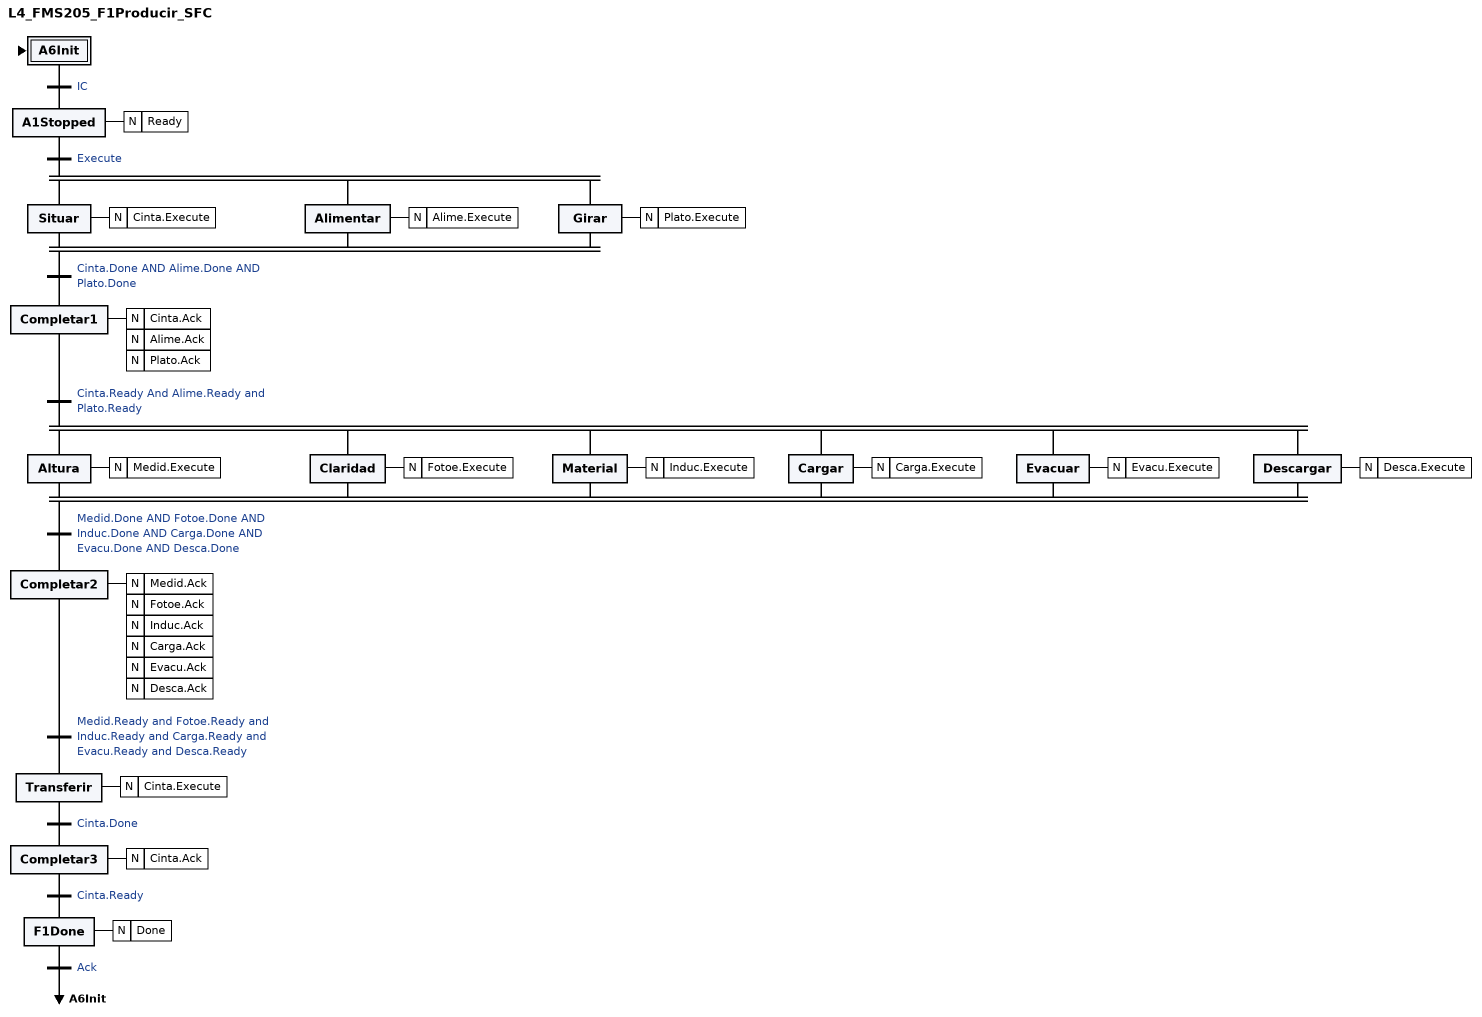
INITIAL_STEP A6Init:
END_STEP
TRANSITION FROM A6Init TO A1Stopped
    := IC;
END_TRANSITION
STEP A1Stopped:
    Ready(N);
END_STEP
TRANSITION FROM A1Stopped TO (Situar, Alimentar, Girar)
    := Execute;
END_TRANSITION
STEP Situar:
    Cinta.Execute(N);
END_STEP
STEP Alimentar:
    Alime.Execute(N);
END_STEP
STEP Girar:
    Plato.Execute(N);
END_STEP
TRANSITION FROM (Situar, Alimentar, Girar) TO Completar1
    := Cinta.Done AND Alime.Done AND Plato.Done;
END_TRANSITION
STEP Completar1:
    Cinta.Ack(N);
    Alime.Ack(N);
    Plato.Ack(N);
END_STEP
TRANSITION FROM Completar1 TO (Altura, Claridad, Material, Cargar, Evacuar, Descargar)
    := Cinta.Ready And Alime.Ready and Plato.Ready;
END_TRANSITION
STEP Altura:
    Medid.Execute(N);
END_STEP
STEP Claridad:
    Fotoe.Execute(N);
END_STEP
STEP Material:
    Induc.Execute(N);
END_STEP
STEP Cargar:
    Carga.Execute(N);
END_STEP
STEP Evacuar:
    Evacu.Execute(N);
END_STEP
STEP Descargar:
    Desca.Execute(N);
END_STEP
TRANSITION FROM (Altura, Claridad, Material, Cargar, Evacuar, Descargar) TO Completar2
    := Medid.Done AND Fotoe.Done AND Induc.Done AND Carga.Done AND Evacu.Done AND Desca.Done;
END_TRANSITION
STEP Completar2:
    Medid.Ack(N);
    Fotoe.Ack(N);
    Induc.Ack(N);
    Carga.Ack(N);
    Evacu.Ack(N);
    Desca.Ack(N);
END_STEP
TRANSITION FROM Completar2 TO Transferir
    := Medid.Ready and Fotoe.Ready and Induc.Ready and Carga.Ready and Evacu.Ready and Desca.Ready;
END_TRANSITION
STEP Transferir:
    Cinta.Execute(N);
END_STEP
TRANSITION FROM Transferir TO Completar3
    := Cinta.Done;
END_TRANSITION
STEP Completar3:
    Cinta.Ack(N);
END_STEP
TRANSITION FROM Completar3 TO F1Done
    := Cinta.Ready;
END_TRANSITION
STEP F1Done:
    Done(N);
END_STEP
TRANSITION FROM F1Done TO A6Init
    := Ack;
END_TRANSITION

END_FUNCTION_BLOCK

// ---- L4 Station Controllers/L4_FMS205_F2SeqPrep_SFC.TcPOU
FUNCTION_BLOCK L4_FMS205_F2SeqPrep_SFC EXTENDS L1_ControllerBase_SFC
// Girar 8 veces el plato para determinar qué tipo de tapa hay en cada sector del plato
VAR_IN_OUT
	Medid			: L3_MedidorTapa;
	Induc		 	: L3_CaptadorInductivo;
	Fotoe			: L3_DetectorFotoelectrico;
	Plato			: L3_PlatoDivisor;
	Tapas			: L6_Tapas;
END_VAR

VAR_OUTPUT
	Seguir 	 		: BOOL;	
	Giros 			: INT;
END_VAR

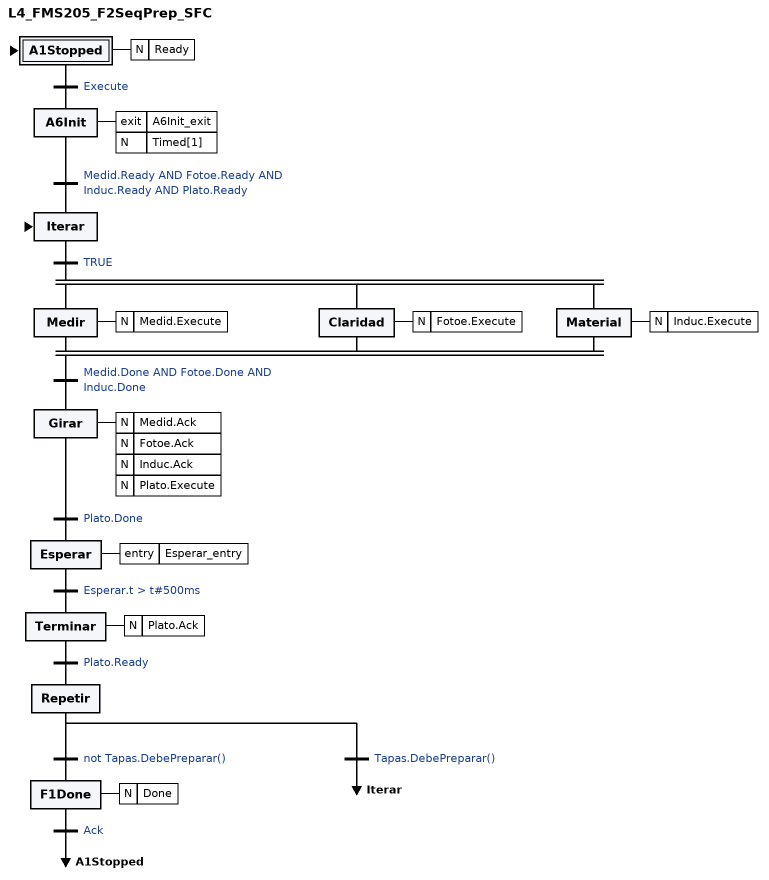
INITIAL_STEP A1Stopped:
    Ready(N);
END_STEP
TRANSITION FROM A1Stopped TO A6Init
    := Execute;
END_TRANSITION
STEP A6Init:
    A6Init_exit(P0);  // exit action
    Timed[1](N);
END_STEP
TRANSITION FROM A6Init TO Iterar
    := Medid.Ready AND Fotoe.Ready AND Induc.Ready AND Plato.Ready;
END_TRANSITION
STEP Iterar:
END_STEP
TRANSITION FROM Iterar TO (Medir, Claridad, Material)
    := TRUE;
END_TRANSITION
STEP Medir:
    Medid.Execute(N);
END_STEP
STEP Claridad:
    Fotoe.Execute(N);
END_STEP
STEP Material:
    Induc.Execute(N);
END_STEP
TRANSITION FROM (Medir, Claridad, Material) TO Girar
    := Medid.Done AND Fotoe.Done AND Induc.Done;
END_TRANSITION
STEP Girar:
    Medid.Ack(N);
    Fotoe.Ack(N);
    Induc.Ack(N);
    Plato.Execute(N);
END_STEP
TRANSITION FROM Girar TO Esperar
    := Plato.Done;
END_TRANSITION
STEP Esperar:
    Esperar_entry(P1);  // entry action
END_STEP
TRANSITION FROM Esperar TO Terminar
    := Esperar.t > t#500ms;
END_TRANSITION
STEP Terminar:
    Plato.Ack(N);
END_STEP
TRANSITION FROM Terminar TO Repetir
    := Plato.Ready;
END_TRANSITION
STEP Repetir:
END_STEP
TRANSITION FROM Repetir TO F1Done
    := not Tapas.DebePreparar();
END_TRANSITION
TRANSITION FROM Repetir TO Iterar
    := Tapas.DebePreparar();
END_TRANSITION
STEP F1Done:
    Done(N);
END_STEP
TRANSITION FROM F1Done TO A1Stopped
    := Ack;
END_TRANSITION

ACTION A6Init_exit:
Giros:=0;
END_ACTION

ACTION Esperar_entry:
Giros:=Giros+1;
END_ACTION

END_FUNCTION_BLOCK

// ---- L4 Station Controllers/L4_FMS205_F3SeqFin_SFC.TcPOU
FUNCTION_BLOCK L4_FMS205_F3SeqFin_SFC EXTENDS L1_ControllerBase_SFC
// Girar 8 veces el plato para determinar qué tipo de tapa hay en cada sector del plato
VAR_INPUT
	TapasOk			: BOOL;
END_VAR

VAR_IN_OUT
	Evacu		 	: L3_Evacuador;
	Plato			: L3_PlatoDivisor;
END_VAR

VAR_OUTPUT
	InitTapas		: BOOL;
	Giros 			: INT := 0;
END_VAR

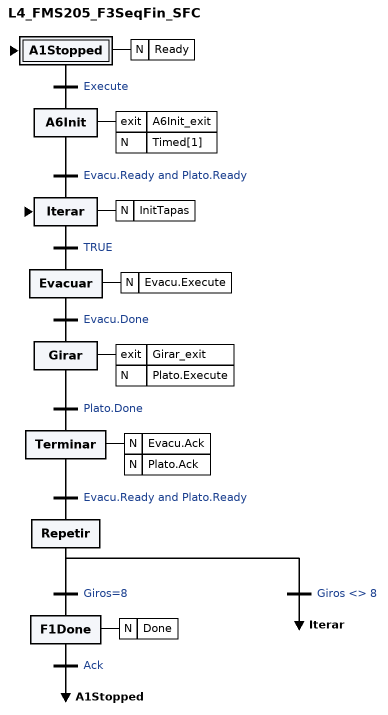
INITIAL_STEP A1Stopped:
    Ready(N);
END_STEP
TRANSITION FROM A1Stopped TO A6Init
    := Execute;
END_TRANSITION
STEP A6Init:
    A6Init_exit(P0);  // exit action
    Timed[1](N);
END_STEP
TRANSITION FROM A6Init TO Iterar
    := Evacu.Ready and Plato.Ready;
END_TRANSITION
STEP Iterar:
    InitTapas(N);
END_STEP
TRANSITION FROM Iterar TO Evacuar
    := TRUE;
END_TRANSITION
STEP Evacuar:
    Evacu.Execute(N);
END_STEP
TRANSITION FROM Evacuar TO Girar
    := Evacu.Done;
END_TRANSITION
STEP Girar:
    Girar_exit(P0);  // exit action
    Plato.Execute(N);
END_STEP
TRANSITION FROM Girar TO Terminar
    := Plato.Done;
END_TRANSITION
STEP Terminar:
    Evacu.Ack(N);
    Plato.Ack(N);
END_STEP
TRANSITION FROM Terminar TO Repetir
    := Evacu.Ready and Plato.Ready;
END_TRANSITION
STEP Repetir:
END_STEP
TRANSITION FROM Repetir TO F1Done
    := Giros=8;
END_TRANSITION
TRANSITION FROM Repetir TO Iterar
    := Giros <> 8;
END_TRANSITION
STEP F1Done:
    Done(N);
END_STEP
TRANSITION FROM F1Done TO A1Stopped
    := Ack;
END_TRANSITION

ACTION A6Init_exit:
Giros:=0;
END_ACTION

ACTION Girar_exit:
Giros:=Giros+1;
END_ACTION

END_FUNCTION_BLOCK

// ---- L4 Station Controllers/L4_FMS205_F6Prueba_SFC.TcPOU
FUNCTION_BLOCK L4_FMS205_F6Prueba_SFC EXTENDS L1_ControllerBase_SFC

VAR_IN_OUT
	Alime			: L3_Alimentador;
	Carga		 	: L3_PickAndPlace;
	Medid			: L3_MedidorTapa;
	Induc		 	: L3_CaptadorInductivo;
	Fotoe			: L3_DetectorFotoelectrico;
	Evacu		 	: L3_Evacuador;
	Desca			: L3_PickAndPlace;
	Plato			: L3_PlatoDivisor;
	Cinta			: L3_Cinta;
END_VAR

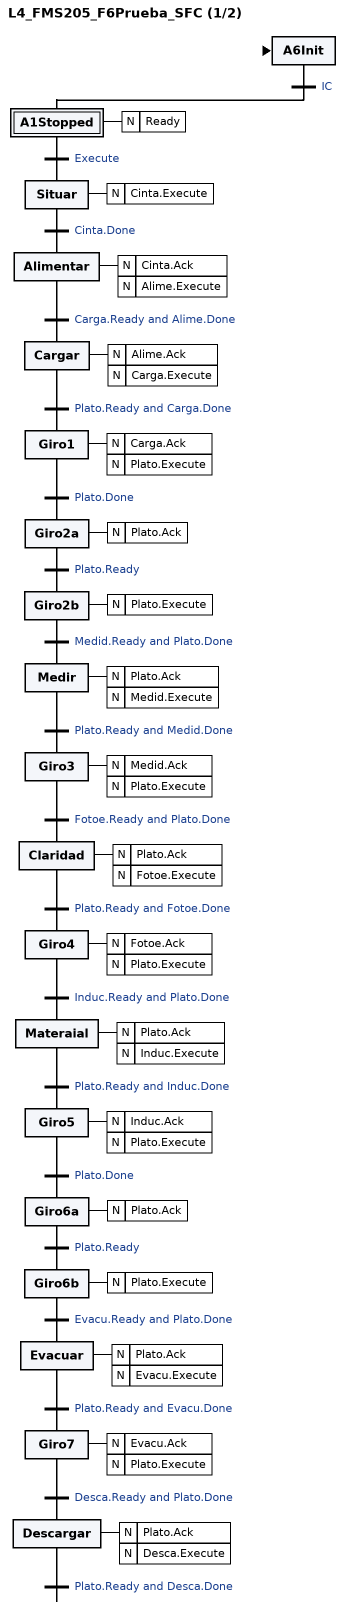
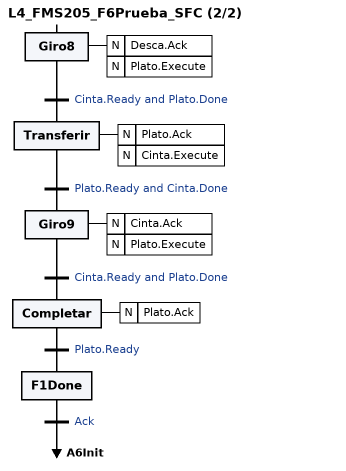
STEP A6Init:
END_STEP
TRANSITION FROM A6Init TO A1Stopped
    := IC;
END_TRANSITION
INITIAL_STEP A1Stopped:
    Ready(N);
END_STEP
TRANSITION FROM A1Stopped TO Situar
    := Execute;
END_TRANSITION
STEP Situar:
    Cinta.Execute(N);
END_STEP
TRANSITION FROM Situar TO Alimentar
    := Cinta.Done;
END_TRANSITION
STEP Alimentar:
    Cinta.Ack(N);
    Alime.Execute(N);
END_STEP
TRANSITION FROM Alimentar TO Cargar
    := Carga.Ready and Alime.Done;
END_TRANSITION
STEP Cargar:
    Alime.Ack(N);
    Carga.Execute(N);
END_STEP
TRANSITION FROM Cargar TO Giro1
    := Plato.Ready and Carga.Done;
END_TRANSITION
STEP Giro1:
    Carga.Ack(N);
    Plato.Execute(N);
END_STEP
TRANSITION FROM Giro1 TO Giro2a
    := Plato.Done;
END_TRANSITION
STEP Giro2a:
    Plato.Ack(N);
END_STEP
TRANSITION FROM Giro2a TO Giro2b
    := Plato.Ready;
END_TRANSITION
STEP Giro2b:
    Plato.Execute(N);
END_STEP
TRANSITION FROM Giro2b TO Medir
    := Medid.Ready and Plato.Done;
END_TRANSITION
STEP Medir:
    Plato.Ack(N);
    Medid.Execute(N);
END_STEP
TRANSITION FROM Medir TO Giro3
    := Plato.Ready and Medid.Done;
END_TRANSITION
STEP Giro3:
    Medid.Ack(N);
    Plato.Execute(N);
END_STEP
TRANSITION FROM Giro3 TO Claridad
    := Fotoe.Ready and Plato.Done;
END_TRANSITION
STEP Claridad:
    Plato.Ack(N);
    Fotoe.Execute(N);
END_STEP
TRANSITION FROM Claridad TO Giro4
    := Plato.Ready and Fotoe.Done;
END_TRANSITION
STEP Giro4:
    Fotoe.Ack(N);
    Plato.Execute(N);
END_STEP
TRANSITION FROM Giro4 TO Materaial
    := Induc.Ready and Plato.Done;
END_TRANSITION
STEP Materaial:
    Plato.Ack(N);
    Induc.Execute(N);
END_STEP
TRANSITION FROM Materaial TO Giro5
    := Plato.Ready and Induc.Done;
END_TRANSITION
STEP Giro5:
    Induc.Ack(N);
    Plato.Execute(N);
END_STEP
TRANSITION FROM Giro5 TO Giro6a
    := Plato.Done;
END_TRANSITION
STEP Giro6a:
    Plato.Ack(N);
END_STEP
TRANSITION FROM Giro6a TO Giro6b
    := Plato.Ready;
END_TRANSITION
STEP Giro6b:
    Plato.Execute(N);
END_STEP
TRANSITION FROM Giro6b TO Evacuar
    := Evacu.Ready and Plato.Done;
END_TRANSITION
STEP Evacuar:
    Plato.Ack(N);
    Evacu.Execute(N);
END_STEP
TRANSITION FROM Evacuar TO Giro7
    := Plato.Ready and Evacu.Done;
END_TRANSITION
STEP Giro7:
    Evacu.Ack(N);
    Plato.Execute(N);
END_STEP
TRANSITION FROM Giro7 TO Descargar
    := Desca.Ready and Plato.Done;
END_TRANSITION
STEP Descargar:
    Plato.Ack(N);
    Desca.Execute(N);
END_STEP
TRANSITION FROM Descargar TO Giro8
    := Plato.Ready and Desca.Done;
END_TRANSITION
STEP Giro8:
    Desca.Ack(N);
    Plato.Execute(N);
END_STEP
TRANSITION FROM Giro8 TO Transferir
    := Cinta.Ready and Plato.Done;
END_TRANSITION
STEP Transferir:
    Plato.Ack(N);
    Cinta.Execute(N);
END_STEP
TRANSITION FROM Transferir TO Giro9
    := Plato.Ready and Cinta.Done;
END_TRANSITION
STEP Giro9:
    Cinta.Ack(N);
    Plato.Execute(N);
END_STEP
TRANSITION FROM Giro9 TO Completar
    := Cinta.Ready and Plato.Done;
END_TRANSITION
STEP Completar:
    Plato.Ack(N);
END_STEP
TRANSITION FROM Completar TO F1Done
    := Plato.Ready;
END_TRANSITION
STEP F1Done:
END_STEP
TRANSITION FROM F1Done TO A6Init
    := Ack;
END_TRANSITION

END_FUNCTION_BLOCK

// ---- L6 Station/L6_FMS205.TcPOU
FUNCTION_BLOCK L6_FMS205 // EXTENDS L1_ModuleBase;

VAR_INPUT
	fbPanel					: L5_Panel := (dr := dr);	
END_VAR

VAR
	// Director, panel y tapas
	dr						: L1_Director;
	tapas					: L6_Tapas;
	
	// módulos de la FMS205
	mdAlimentador			: L3_Alimentador			:= (dr:=dr, ID := 1, Name := 'Alimentador');
	mdPickAndPlaceCarga 	: L3_PickAndPlace			:= (dr:=dr, ID := 2, Name := 'Carga');
	mdMedidorTapa			: L3_MedidorTapa			:= (dr:=dr, ID := 3, Name := 'Medidor');
	mdCaptadorInductivo 	: L3_CaptadorInductivo		:= (dr:=dr, ID := 4, Name := 'Inductivo');
	mdDetectorFotoelectrico : L3_DetectorFotoelectrico	:= (dr:=dr, ID := 5, Name := 'Fotoeléctrico');
	mdEvacuador			 	: L3_Evacuador				:= (dr:=dr, ID := 6, Name := 'Evacuador');
	mdPickAndPlaceDescarga 	: L3_PickAndPlace			:= (dr:=dr, ID := 7, Name := 'Descarga');
	mdPlatoDivisor			: L3_PlatoDivisor			:= (dr:=dr, ID := 8, Name := 'Plato');
	mdCinta					: L3_Cinta					:= (dr:=dr, ID := 9, Name := 'Cinta');
	
	// controladores a nivel estación
	ctrlF1Producir			: L4_FMS205_F1Producir_SFC; 
	ctrlF2SeqPrep			: L4_FMS205_F2SeqPrep_SFC;		
	ctrlF3SeqFin			: L4_FMS205_F3SeqFin_SFC;		
	ctrlF6Prueba			: L4_FMS205_F6Prueba_SFC;
END_VAR

METHOD InitialConditions : BOOL
(* La estación está en condiciones iniciales si cada módulo lo está *)
InitialConditions := (
		mdAlimentador.IC AND
		mdPickAndPlaceCarga.IC AND
		mdMedidorTapa.IC AND 
		mdCaptadorInductivo.IC AND
		mdDetectorFotoelectrico.IC AND
		mdEvacuador.IC AND
		mdPickAndPlaceDescarga.IC AND
		mdPlatoDivisor.IC AND
		mdCinta.IC )  OR dr.gmLocalHost;
END_METHOD

METHOD IsFailied : BOOL
VAR
	NumError	: UDINT;
	Mensaje		: string;
END_VAR
IsFailied:=TRUE;	
IF dr.gmModeActual = L1_GEMMA.A6Inicializando THEN
	IsFailied:=FALSE;
	ManageErrors();
ELSIF dr.gmModeActual = L1_GEMMA.A5PreparandoTrasFallo OR dr.gmModeActual=L1_GEMMA.D2TratamientoFallos THEN
	IF mdAlimentador.fbController.NumError <> 0 THEN
		Mensaje := 'Fallo en alimentador, error=';
		NumError :=	mdAlimentador.fbController.NumError;
		
	ELSIF mdPickAndPlaceCarga.fbController.NumError <> 0 THEN
		Mensaje := 'Fallo en brazo de carga, error=';
		NumError := mdPickAndPlaceCarga.fbController.NumError; 
		
	ELSIF mdMedidorTapa.fbController.NumError <> 0 THEN
		Mensaje := 'Fallo en medidor de altura, error=';
		NumError := mdMedidorTapa.fbController.NumError;
		
	ELSIF mdDetectorFotoelectrico.fbController.NumError <> 0 THEN
		Mensaje := 'Fallo en detector fotoeléctrico, error=';
		NumError := mdDetectorFotoelectrico.fbController.NumError;
		
	ELSIF mdCaptadorInductivo.fbController.NumError<>0 THEN
		Mensaje := 'Fallo en captador inductivo, error=';
		NumError := mdCaptadorInductivo.fbController.NumError;
	
	ELSIF mdEvacuador.fbController.NumError <> 0 THEN
		Mensaje := 'Fallo en evacuador, error=';
		NumError := mdEvacuador.fbController.NumError;
		
	ELSIF  mdPickAndPlaceDescarga.fbController.NumError <> 0 THEN
		Mensaje := 'Fallo en brazo de descarga, error=';
		NumError := mdPickAndPlaceDescarga.fbController.NumError;
		
	ELSIF mdPlatoDivisor.fbController.NumError <> 0 THEN
		Mensaje := 'Fallo en plato giratorio, error=';
		NumError := mdPlatoDivisor.fbController.NumError;
		
	ELSIF mdCinta.fbController.NumError <> 0 THEN
		Mensaje := 'Fallo en cinta, error=';
		NumError := mdCinta.fbController.NumError;
	
	ELSE
		fbPanel.swMensaje := '';
		IsFailied := FALSE;
	END_IF
	
	IF IsFailied THEN
		fbPanel.swMensaje := CONCAT(Mensaje, TO_STRING(NumError));
	END_IF

ELSE
	IsFailied:=FALSE;		
END_IF
END_METHOD

METHOD IsPaused : BOOL
VAR_INPUT
END_VAR
IsPaused := 
		mdAlimentador.fbController.IsPaused() AND
		mdPickAndPlaceCarga.fbController.IsPaused() AND
		mdMedidorTapa.fbController.IsPaused() AND 
		mdCaptadorInductivo.fbController.IsPaused() AND
		mdDetectorFotoelectrico.fbController.IsPaused() AND
		mdEvacuador.fbController.isPaused() AND
		mdPickAndPlaceDescarga.fbController.IsPaused() AND
		mdPlatoDivisor.fbController.IsPaused() AND
		mdCinta.fbController.IsPaused(); (* AND
		ctrlF1Producir.IsPaused() AND
		ctrlF2SeqPrep.IsPaused() AND
		ctrlF3SeqFin.IsPaused() AND
		ctrlF6Prueba.IsPaused();*)
END_METHOD

METHOD ManageErrors : BOOL
mdAlimentador.fbController.ResetError();
mdAlimentador.fbController.ResetError();
mdPickAndPlaceCarga.fbController.ResetError();
mdMedidorTapa.fbController.ResetError();
mdCaptadorInductivo.fbController.ResetError();
mdDetectorFotoelectrico.fbController.ResetError();
mdEvacuador.fbController.ResetError();
mdPickAndPlaceDescarga.fbController.ResetError();
mdPlatoDivisor.fbController.ResetError();
mdCinta.fbController.ResetError();
ctrlF1Producir.ResetError();
ctrlF2SeqPrep.ResetError();
ctrlF3SeqFin.ResetError();
ctrlF6Prueba.ResetError();
END_METHOD

METHOD ProcessCycle : BOOL
// calcular consignas en función del panel y del modo Gemma
dr.Failure 									:= IsFailied();
fbPanel.ProcessCycle(dr:=dr, gmModeActual := dr.gmModeActual, tmReinicio := dr.tmTiempoReinicio);
dr.ProcessCycle(); 

// ejecutar el ciclo de cada Grafcet a nivel estación
ctrlF1Producir.ProcessCycle(dr.gmModeActual);					
ctrlF2SeqPrep.ProcessCycle(dr.gmModeActual);
ctrlF3SeqFin.ProcessCycle(dr.gmModeActual);
ctrlF6Prueba.ProcessCycle(dr.gmModeActual);

// decidir qué tiene que hacer cada módulo
mdAlimentador.Alimentar					:= NOT dr.EndBatch AND NOT tapas.EstaAlimentada; // mdAlimentador.TapaAlimentada;
mdPickAndPlaceCarga.Mover				:= NOT dr.EndBatch AND tapas.EstaAlimentada AND tapas.PuedeCargar(); //  mdAlimentador.TapaAlimentada 
//IF mdPickAndPlaceCarga.TapaMovida THEN
	//mdAlimentador.TapaAlimentada		:= FALSE;
	//tapas.EstaAlimentada				:= FALSE;
	//mdPickAndPlaceCarga.TapaMovida		:= FALSE;	
//END_IF

mdMedidorTapa.Medir						:= tapas.DebeMedir();
mdEvacuador.Evacuar						:= tapas.PuedeEvacuar(gmMode:=dr.gmModeActual);
mdPickAndPlaceDescarga.Mover			:= NOT dr.EndBatch AND mdCinta.Carro_Situado AND tapas.PuedeDescargar();
//IF mdPickAndPlaceDescarga.TapaMovida THEN
	//mdCinta.TapaDescargada				:= TRUE;
	//mdCinta.Transferir					:= TRUE;
	//mdPickAndPlaceDescarga.TapaMovida	:= FALSE;
//END_IF


// controlar el flujo a nivel de la estación
CASE dr.gmModeActual OF
	L1_GEMMA.A1ParadaInicial:						// esperar a que se pida hacer altgo
		dr.EndCycle	:= FALSE;
		dr.EndBatch	:= FALSE;		

	//L1_GEMMA.A3ParadaEstado: 						// esperar la puesta en marcha o reanudar tras parada		
	//L1_GEMMA.A4ParadaObtenida:
	//	dr.IsPaused := IsPaused(); 

	L1_GEMMA.A5PreparandoTrasFallo:
		ManageErrors();		

	L1_GEMMA.A6Inicializando:
		dr.Failure						:= FALSE;
		dr.IsPaused						:= FALSE;
		dr.IC							:= InitialConditions();
		tapas.Inicializar();		
		
	L1_GEMMA.D1ParadaEmergencia:
		dr.IC							:= FALSE;	// obliga a ejecutar la inicialización
		
	L1_GEMMA.D2TratamientoFallos:					// esperar a que el usuario arregle el error
		dr.Failure 		:= IsFailied(); 			// redundante. ManageErrors(); ?
		
	L1_GEMMA.F1ProduccionNormal,
	L1_GEMMA.A2ParaFinCiclo:
		ctrlF1Producir.IC 				:= InitialConditions();
		dr.EndCycle 					:= ctrlF1Producir.Done;
		IF ctrlF1Producir.Done THEN
			dr.EndCycle					:= TRUE;
			dr.cnA3_Estado				:= dr.cnA2_FinCiclo;
			ctrlF1Producir.Execute		:= FALSE;
			ctrlF1Producir.Ack			:= TRUE;			
			dr.EndBatch 				:= tapas.ResReal >= tapas.ReqNumero;			
		ELSIF ctrlF1Producir.Ready AND NOT dr.EndCycle THEN
			dr.EndCycle					:= FALSE;
			ctrlF1Producir.Execute		:= TRUE;
			ctrlF1Producir.Ack			:= FALSE;
		END_IF
		ctrlF1Producir(	Alime:=mdAlimentador, Carga:=mdPickAndPlaceCarga, Medid:=mdMedidorTapa, 
				Fotoe:=mdDetectorFotoelectrico, Induc:=mdCaptadorInductivo, Evacu:=mdEvacuador,	
				Desca:=mdPickAndPlaceDescarga, Plato:=mdPlatoDivisor, Cinta:=mdCinta);						
	
	L1_GEMMA.F2SecuenciaPreparacion:		
		//ctrlF2SeqPrep.IC				:= InitialConditions();			
		IF ctrlF2SeqPrep.Ready THEN
			ctrlF2SeqPrep.Execute		:= TRUE; // ctrlF2SeqPrep.Ready;
			ctrlF2SeqPrep.Ack			:= FALSE;
			//ctrlF2SeqPrep.cnF2_Preparar	:= dr.cnF2_Preparar;
		ELSIF ctrlF2SeqPrep.Done THEN
			dr.cnF2_Preparar		:= FALSE;
			ctrlF2SeqPrep.Execute 	:= FALSE;
			ctrlF2SeqPrep.Ack		:= TRUE;
		END_IF
		ctrlF2SeqPrep(Medid:=mdMedidorTapa, Fotoe:=mdDetectorFotoelectrico, Induc:=mdCaptadorInductivo, Plato:=mdPlatoDivisor);

	L1_GEMMA.F3SecuenciaFinalizacion:
		//ctrlF3SeqFin.IC					:= InitialConditions();
		IF ctrlF3SeqFin.Ready THEN
			ctrlF3SeqFin.Execute 		:= TRUE;
			ctrlF3SeqFin.Ack			:= FALSE;
		ELSIF ctrlF3SeqFin.Done THEN
			dr.cnF3_Finalizar 			:= FALSE;
			ctrlF3SeqFin.Execute 		:= FALSE;
			ctrlF3SeqFin.Ack			:= TRUE;
			dr.cnF1_Producir			:= FALSE;
			dr.cnF2_Preparar			:= FALSE;
			dr.cnF3_Finalizar			:= FALSE;
		END_IF
		ctrlF3SeqFin(Evacu:=mdEvacuador, Plato:=mdPlatoDivisor);	
							
	L1_GEMMA.F4VerificacionSinOrden: 
		IF fbPanel.swF4_Avanza THEN		
			mdCinta.RUN.ForceValue(NewValue:=TRUE);
			mdCinta.REV.ForceValue(NewValue:=FALSE);
		ELSIF fbPanel.swF4_Retroc THEN
			mdCinta.RUN.ForceValue(NewValue:=TRUE);
			mdCinta.REV.ForceValue(NewValue:=TRUE);
		END_IF		

	L1_GEMMA.F5VerificacionOrdenada:
		mdAlimentador.Execute          		:= fbPanel.swF5_Ejecutar AND fbPanel.swF5_Alimentar; 		//tapas.ExeAlime; mdAlimentador.Alimentar AND 
		mdMedidorTapa.Execute          		:= fbPanel.swF5_Ejecutar AND fbPanel.swF5_Medir; 		//tapas.ExeMedid;
		mdDetectorFotoelectrico.Execute		:= fbPanel.swF5_Ejecutar AND fbPanel.swF5_Claridad; 	//  tapas.ExeFotoe;
		mdCaptadorInductivo.Execute    		:= fbPanel.swF5_Ejecutar AND fbPanel.swF5_Material;
		mdPickAndPlaceCarga.Execute			:= fbPanel.swF5_Ejecutar AND fbPanel.swF5_Cargar; 		// AND fbPanel.swF5_Ejecutar;
		mdEvacuador.Execute            		:= fbPanel.swF5_Ejecutar AND fbPanel.swF5_Evacuar;	 	//tapas.ExeEvacu;
		mdPickAndPlaceDescarga.Execute		:= fbPanel.swF5_Ejecutar AND fbPanel.swF5_Descargar;
		mdPlatoDivisor.Execute       		:= fbPanel.swF5_Ejecutar AND fbPanel.swF5_Girar;				
		mdCinta.Execute						:= fbPanel.swF5_Ejecutar AND  
												((mdCinta.Situar AND fbPanel.swF5_Situar ) OR (mdCinta.Transferir AND fbPanel.swF5_Transferir));
		IF NOT mdCinta.Carro_Situado AND fbPanel.swF5_Situar THEN
			mdCinta.Situar						:= TRUE;
			mdCinta.Transferir					:= FALSE;	
		ELSIF mdCinta.Carro_Situado AND NOT mdCinta.Carro_Transfer AND fbPanel.swF5_Transferir THEN
			mdCinta.Situar						:= FALSE;
			mdCinta.Transferir					:= TRUE; 
		END_IF
		mdAlimentador.Ack               := fbPanel.swF5_Ack AND fbPanel.swF5_Alimentar;
		mdPickAndPlaceCarga.Ack         := fbPanel.swF5_Ack AND fbPanel.swF5_Cargar;
		mdMedidorTapa.Ack               := fbPanel.swF5_Ack AND fbPanel.swF5_Medir;
		mdDetectorFotoelectrico.Ack		:= fbPanel.swF5_Ack AND fbPanel.swF5_Claridad;
		mdCaptadorInductivo.Ack         := fbPanel.swF5_Ack AND fbPanel.swF5_Material;
		mdEvacuador.Ack                 := fbPanel.swF5_Ack AND fbPanel.swF5_Evacuar;
		mdPickAndPlaceDescarga.Ack      := fbPanel.swF5_Ack AND fbPanel.swF5_Descargar;
		mdPlatoDivisor.Ack              := fbPanel.swF5_Ack AND fbPanel.swF5_Girar;
		mdCinta.Ack						:= fbPanel.swF5_Ack AND (fbPanel.swF5_Situar OR fbPanel.swF5_Transferir);			
				
	L1_GEMMA.F6Probando:
		ctrlF6Prueba.IC					:= InitialConditions();
		IF ctrlF6Prueba.Ready THEN
			ctrlF6Prueba.Execute 		:= TRUE;
			ctrlF6Prueba.Ack			:= FALSE;
		ELSIF ctrlF6Prueba.Done THEN
			ctrlF6Prueba.Ack			:= TRUE;
			ctrlF6Prueba.Execute		:= FALSE;			
		END_IF			
		ctrlF6Prueba(	Alime:=mdAlimentador, Carga:=mdPickAndPlaceCarga, Medid:=mdMedidorTapa, 
			Fotoe:=mdDetectorFotoelectrico, Induc:=mdCaptadorInductivo, Evacu:=mdEvacuador,	
			Desca:=mdPickAndPlaceDescarga, Plato:=mdPlatoDivisor, Cinta:=mdCinta);
	
END_CASE

mdAlimentador.ProcessCycle				(dr:=dr, tapas:=tapas); // ejecutar el ciclo de cada uno de los módulos
mdPickAndPlaceCarga.ProcessCycle		(dr:=dr, tapas:=tapas);
mdMedidorTapa.ProcessCycle				(dr:=dr, tapas:=tapas);	
mdDetectorFotoelectrico.ProcessCycle	(dr:=dr, tapas:=tapas);
mdCaptadorInductivo.ProcessCycle		(dr:=dr, tapas:=tapas);
mdEvacuador.ProcessCycle				(dr:=dr, tapas:=tapas);
mdPickAndPlaceDescarga.ProcessCycle		(dr:=dr, tapas:=tapas);
mdPlatoDivisor.ProcessCycle				(dr:=dr, tapas:=tapas);
mdCinta.ProcessCycle					(dr:=dr, tapas:=tapas);
tapas.ProcessCycle						(dr:=dr, pn:=fbPanel, NumGiros := mdPlatoDivisor.NumGiros);
END_METHOD

END_FUNCTION_BLOCK

// ---- L6 Station/MAIN.TcPOU
PROGRAM MAIN
VAR
	fbFMS205 : L6_FMS205;	
END_VAR

fbFMS205.ProcessCycle();

END_PROGRAM

// ---- GlobalTextList.TcGTLO
TEXTLIST GlobalTextList
  440 = ' mm'
  584 = '%0.2f'
  209 = '%d'
  1644 = '%f'
  471 = '%s'
  127 = '%S'
  268 = '0=%s'
  50 = '0º'
  53 = '135º'
  54 = '180º'
  55 = '225º'
  56 = '270º'
  57 = '315º'
  51 = '45º'
  52 = '90º'
  208 = 'a0'
  210 = 'a1'
  857 = 'AAIn'
  856 = 'ABIn'
  442 = 'Aceptar Aluminio'
  907 = 'Aceptar aluminio'
  446 = 'Aceptar Blancas'
  932 = 'Aceptar blancas'
  449 = 'Aceptar Negras'
  803 = 'Ack'
  282 = 'AckExecute'
  343 = 'Alimentador'
  225 = 'Alimentar'
  563 = 'AlturaMm'
  562 = 'AlturaOut'
  920 = 'Alu. Alta'
  913 = 'Alu. Baja'
  855 = 'Aluminio'
  863 = 'AS'
  447 = 'Avanza'
  421 = 'Avisador sonoro'
  206 = 'A_1'
  212 = 'b0'
  213 = 'b1'
  862 = 'BAIn'
  861 = 'BBIn'
  860 = 'Blanco'
  945 = 'Bln. Alta'
  939 = 'Bln. Baja'
  211 = 'B_1'
  320 = 'Carga'
  559 = 'Cargar'
  451 = 'Cinta'
  267 = 'Claridad'
  521 = 'Color'
  566 = 'ColorOut'
  1494 = 'Conmutador encendido/apagado'
  491 = 'Continuar'
  475 = 'cp0'
  483 = 'cp1'
  499 = 'cp2'
  216 = 'C_1'
  610 = 'd0'
  285 = 'Descarga'
  599 = 'Descargar'
  49 = 'Descripción modo'
  746 = 'Det. Fotoeléctrico'
  750 = 'Det. Inductivo'
  565 = 'DetColor'
  571 = 'DetMaterial'
  221 = 'df'
  218 = 'dh'
  222 = 'di'
  865 = 'DPO'
  604 = 'D_1'
  487 = 'Ejecutar'
  215 = 'Emerg'
  731 = 'Emergencia (D1)'
  214 = 'Empezar'
  717 = 'Empezar (F1)'
  205 = 'Estacion'
  390 = 'Estación'
  2182 = 'Estación (F6)'
  24 = 'Evacuador'
  1256 = 'Evacuar'
  699 = 'EvacuarRechazar'
  514 = 'Execute'
  439 = 'E_1'
  703 = 'F+'
  266 = 'F-'
  797 = 'f0'
  780 = 'f1'
  349 = 'Fin Ciclo (A2)'
  1159 = 'Fin Ciclo (A2)(F3)'
  885 = 'Fin ciclo A2'
  873 = 'Finalizar (F3)'
  226 = 'FM'
  386 = 'FMS205 - Estación de carga de tapas'
  1269 = 'FMS205 - Estación de carga de tapas       -       Equipo G07 Patos Descartados'
  207 = 'Fotoelectrico'
  223 = 'Funcion'
  755 = 'Función (F5)'
  48 = 'Fx'
  224 = 'F_0'
  227 = 'F_1'
  257 = 'G+'
  19 = 'g0'
  615 = 'Girar'
  560 = 'G_1'
  568 = 'h0'
  569 = 'h1'
  567 = 'H_1'
  576 = 'i0'
  582 = 'i1'
  352 = 'Inductivo'
  688 = 'Inicializar (A6)'
  573 = 'I_1'
  593 = 'J_1'
  202 = 'k1'
  201 = 'K_1'
  866 = 'LA'
  203 = 'Llenar'
  722 = 'Llenar (F2)'
  864 = 'LM'
  6 = 'Logo'
  217 = 'L_1'
  888 = 'Lámpara de alarma'
  791 = 'Lámpara de marcha'
  78 = 'MAIN.fbFMS205.fbPanel.ttPE_Seta'
  1352 = 'Marcha'
  1121 = 'Material'
  572 = 'MaterialOut'
  775 = 'Medidor'
  1334 = 'Medir Altura'
  561 = 'MedirAlt'
  515 = 'MensajesOut'
  816 = 'Metalica'
  503 = 'Modo'
  511 = 'ModoDesc'
  507 = 'ModoOut'
  869 = 'NAIn'
  868 = 'NBIn'
  664 = 'NegarSensores'
  867 = 'Negro'
  712 = 'Ngr. Alta'
  708 = 'Ngr. Baja'
  11 = 'NoTapas'
  842 = 'NoTapasIn'
  1279 = 'Número de Tapas'
  900 = 'Número de tapas'
  228 = 'Panel'
  377 = 'Panel de pruebas'
  894 = 'Panel Físico'
  9 = 'PanelFisico'
  854 = 'PanelImagen'
  1717 = 'Parada ciclo (A2)'
  1709 = 'Parada ciclo A2'
  2043 = 'Parada de emergencia (A1)'
  1328 = 'Parada de Emergencia (D1)'
  1073 = 'Parada estado (A3)'
  1473 = 'Pausa (A3)'
  872 = 'Pausa A3'
  219 = 'Pausar'
  62 = 'Pausar (A3)'
  736 = 'Pausar (A3->4)'
  1401 = 'Pausar (á3)'
  1186 = 'Pausar A3'
  1155 = 'Pausr (á3)'
  845 = 'PE'
  843 = 'Pendientes'
  844 = 'PendientesIn'
  870 = 'Planta'
  926 = 'Planta (F4)'
  660 = 'Plato'
  847 = 'PM'
  846 = 'POC'
  459 = 'pp'
  1761 = 'Preparar (F2)'
  1462 = 'Probar (F6)'
  1491 = 'Probar ciclo en serie (F6)'
  1903 = 'Probar Estación (F6)'
  1861 = 'Producción'
  1733 = 'Producción normal'
  1320 = 'Producir (F1)'
  292 = 'Producir aluminio'
  871 = 'Producir blancas'
  1521 = 'Producir Negras'
  737 = 'Prueba serie (F6)'
  294 = 'Pruebas (F6)'
  1484 = 'PS'
  1094 = 'Pulsador de inicializar (A6)'
  764 = 'Pulsador de marcha'
  445 = 'Pulsador de parada'
  852 = 'Realizadas'
  853 = 'RealizadasOut'
  828 = 'Reanudar'
  316 = 'Reanudar (F1)'
  858 = 'Rechazadas'
  859 = 'RechazadasOut'
  587 = 'Rechazar'
  7 = 'Requisitos'
  389 = 'Requisitos de producción'
  220 = 'Reset'
  1263 = 'Reset (A6)'
  741 = 'Reset (A6->1)'
  8 = 'Resultados'
  47 = 'Retroc.'
  467 = 'Retrocede'
  472 = 'REV'
  455 = 'RUN'
  479 = 'R_1'
  263 = 'Selector manual (F4) automático'
  995 = 'Selector manual automático (F4)'
  443 = 'Situar'
  848 = 'SM'
  570 = 'Speed'
  495 = 'S_1'
  674 = 'Test'
  5 = 'Titulo'
  762 = 'TK_1'
  70 = 'tooltip generada'
  463 = 'Transferir'
  849 = 'Umbral'
  436 = 'Umbral Alta/Baja'
  850 = 'UmbralIn'
  851 = 'UmbralMm'
  738 = 'V+'
  790 = 'v1'
  204 = 'Vaciar'
  727 = 'Vaciar (F3)'
  10 = 'Velocidad'
  879 = 'Verificar Función (F5)'
  1321 = 'Verificar Planta (F4)'
  1336 = 'Visto'
  681 = 'VistoContinuar'
  564 = 'V_1'
  383 = 'xx'
END_TEXTLIST

// ---- L5 Station User Interfaces/L5_FMS205VISU.TcVIS
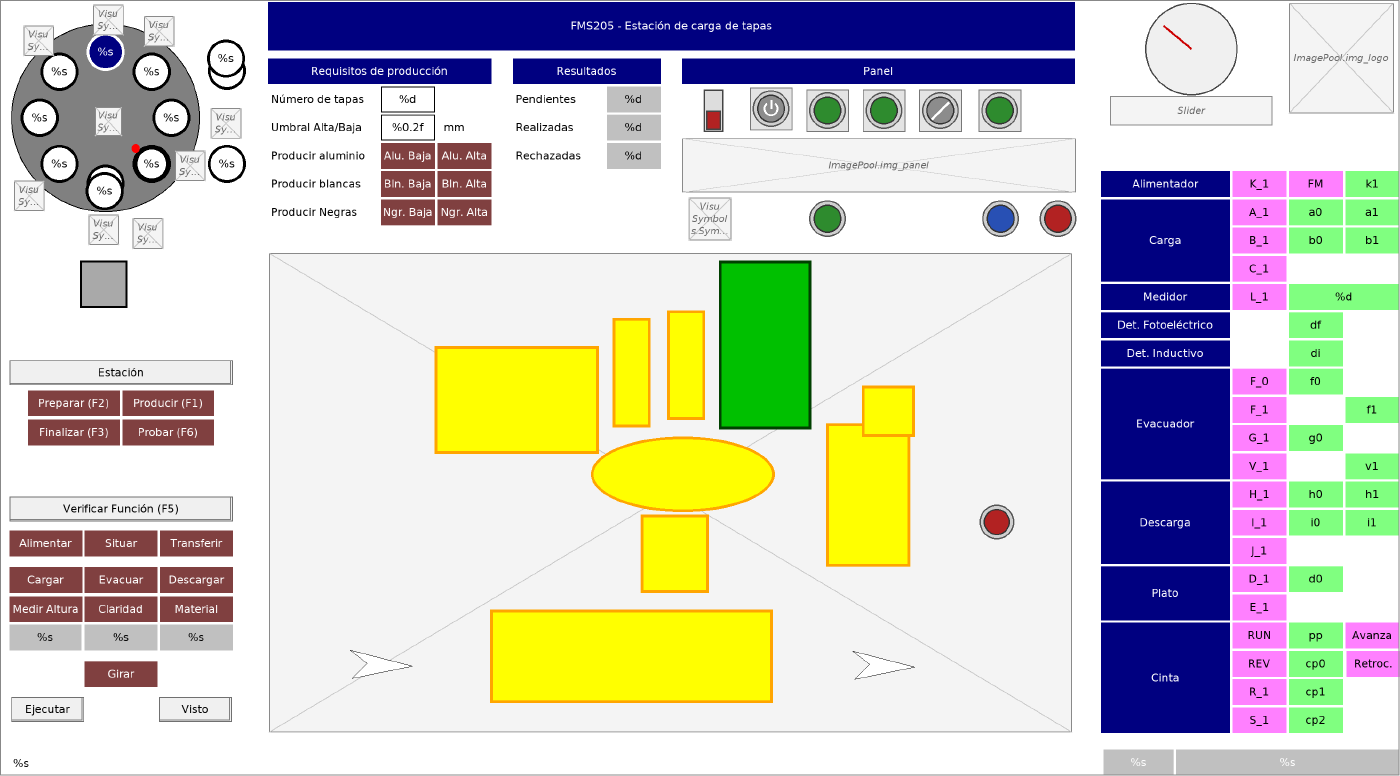
VISUALIZATION L5_FMS205VISU  // 1488x825
    Rectangle (285,2 857x51), "FMS205 - Estación de carga de tapas", colour variable: MAIN.fbFMS205.dr.gmModeColor
        p3450524324: MAIN.fbFMS205.dr.gmModeColor
    Rectangle (285,62 237x27), "Requisitos de producción"
    Rectangle (545,62 157x27), "Resultados"
    Rectangle (725,62 417x27), "Panel"
    Rectangle (285,92 157x27), "Número de tapas"
    Rectangle (405,92 57x27), "%d", text variable: MAIN.fbFMS205.tapas.ReqNumero
        OnMouseClick: write the text variable via VisuDialogs.Numpad, min 1, max 500
    Rectangle (545,92 97x27), "Pendientes"
    Rectangle (645,92 57x27), "%d", text variable: MAIN.fbFMS205.tapas.ResPend
    Rectangle (285,122 117x27), "Umbral Alta/Baja"
    Rectangle (405,122 57x27), "%0.2f", text variable: MAIN.fbFMS205.tapas.ReqAlta
        p4168582468: 'Atura en mm mínima para considerar que la tapa es alta'
        OnMouseClick: write the text variable via VisuDialogs.Numpad, min 2, max 5
    Rectangle (465,122 37x27), "mm"
    Rectangle (545,122 117x27), "Realizadas"
    Rectangle (645,122 57x27), "%d", text variable: MAIN.fbFMS205.tapas.ResReal
    Rectangle (285,152 117x27), "Producir aluminio"
    Rectangle (405,152 57x27), "Alu. Baja"
        toggle MAIN.fbFMS205.tapas.ReqAluBaja
    Rectangle (465,152 57x27), "Alu. Alta"
        toggle MAIN.fbFMS205.tapas.ReqAluAlta
    Rectangle (545,152 117x27), "Rechazadas"
    Rectangle (645,152 57x27), "%d", text variable: MAIN.fbFMS205.tapas.ResRech
    Rectangle (285,182 117x27), "Producir blancas"
    Rectangle (405,182 57x27), "Bln. Baja"
        toggle MAIN.fbFMS205.tapas.ReqBlnBaja
    Rectangle (465,182 57x27), "Bln. Alta"
        toggle MAIN.fbFMS205.tapas.ReqBlnAlta
    Rectangle (1170,182 137x27), "Alimentador", input disabled if: not MAIN.fbFMS205.dr.cnF4_Planta
    Rectangle (1310,182 57x27), "K_1", input disabled if: not MAIN.fbFMS205.dr.cnF4_Planta
        toggle MAIN.fbFMS205.mdAlimentador.K_1.uiValue
    Rectangle (1370,182 57x27), "FM", input disabled if: not MAIN.fbFMS205.dr.cnF4_Planta
        toggle MAIN.fbFMS205.mdAlimentador.FM.uiValue
    Rectangle (1430,182 57x27), "k1", input disabled if: not MAIN.fbFMS205.dr.cnF4_Planta
        toggle MAIN.fbFMS205.mdAlimentador.k1.uiValue
    Rectangle (285,212 117x27), "Producir Negras"
    Rectangle (405,212 57x27), "Ngr. Baja"
        toggle MAIN.fbFMS205.tapas.ReqNgrBaja
    Rectangle (465,212 57x27), "Ngr. Alta"
        toggle MAIN.fbFMS205.tapas.ReqNgrAlta
    Rectangle (1170,212 137x87), "Carga", input disabled if: not MAIN.fbFMS205.dr.cnF4_Planta
    Rectangle (1310,212 57x27), "A_1", input disabled if: not MAIN.fbFMS205.dr.cnF4_Planta
        toggle MAIN.fbFMS205.mdPickAndPlaceCarga.HOR.uiValue
    Rectangle (1370,212 57x27), "a0", input disabled if: not MAIN.fbFMS205.dr.cnF4_Planta
        toggle MAIN.fbFMS205.mdPickAndPlaceCarga.h0.uiValue
    Rectangle (1430,212 57x27), "a1", input disabled if: not MAIN.fbFMS205.dr.cnF4_Planta
        toggle MAIN.fbFMS205.mdPickAndPlaceCarga.h1.uiValue
    Rectangle (1310,242 57x27), "B_1", input disabled if: not MAIN.fbFMS205.dr.cnF4_Planta
        toggle MAIN.fbFMS205.mdPickAndPlaceCarga.VER.uiValue
    Rectangle (1370,242 57x27), "b0", input disabled if: not MAIN.fbFMS205.dr.cnF4_Planta
        toggle MAIN.fbFMS205.mdPickAndPlaceCarga.v0.uiValue
    Rectangle (1430,242 57x27), "b1", input disabled if: not MAIN.fbFMS205.dr.cnF4_Planta
        toggle MAIN.fbFMS205.mdPickAndPlaceCarga.v1.uiValue
    Rectangle (286,269 837x507), "Estacion"
    Rectangle (30,415 97x27), "Preparar (F2)", input disabled if: not MAIN.fbFMS205.fbPanel.mdF1Producir
        toggle MAIN.fbFMS205.fbPanel.swF2_Preparar
    Rectangle (130,415 97x27), "Producir (F1)", input disabled if: not MAIN.fbFMS205.fbPanel.mdF1Producir
        toggle MAIN.fbFMS205.fbPanel.swF1_Producir
    Rectangle (1310,272 57x27), "C_1", input disabled if: not MAIN.fbFMS205.dr.cnF4_Planta
        toggle MAIN.fbFMS205.mdPickAndPlaceCarga.PIN.uiValue
    Rectangle (1170,302 137x27), "Medidor", input disabled if: not MAIN.fbFMS205.dr.cnF4_Planta
    Rectangle (1310,302 57x27), "L_1", input disabled if: not MAIN.fbFMS205.dr.cnF4_Planta
        toggle MAIN.fbFMS205.mdMedidorTapa.L_1.uiValue
    Rectangle (1370,302 117x27), "%d", text variable: MAIN.fbFMS205.mdMedidorTapa.dh, input disabled if: not MAIN.fbFMS205.dr.cnF4_Planta
    Rectangle (1170,332 137x27), "Det. Fotoeléctrico", input disabled if: not MAIN.fbFMS205.dr.cnF4_Planta
    Rectangle (1370,332 57x27), "df", input disabled if: not MAIN.fbFMS205.dr.cnF4_Planta
        toggle MAIN.fbFMS205.mdDetectorFotoelectrico.df.uiValue
    Rectangle (1170,362 137x27), "Det. Inductivo", input disabled if: not MAIN.fbFMS205.dr.cnF4_Planta
    Rectangle (1370,362 57x27), "di", input disabled if: not MAIN.fbFMS205.dr.cnF4_Planta
        toggle MAIN.fbFMS205.mdCaptadorInductivo.di.uiValue
    Rectangle (1170,392 137x117), "Evacuador", input disabled if: not MAIN.fbFMS205.dr.cnF4_Planta
    Rectangle (1310,392 57x27), "F_0", input disabled if: not MAIN.fbFMS205.dr.cnF4_Planta
        toggle MAIN.fbFMS205.mdEvacuador.F_0.uiValue
    Rectangle (1370,392 57x27), "f0", input disabled if: not MAIN.fbFMS205.dr.cnF4_Planta
        toggle MAIN.fbFMS205.mdEvacuador.f0.uiValue
    Button (10,528 237x26), "Verificar Función (F5)", input disabled if: not (MAIN.fbFMS205.dr.gmModeActual=L1_GEMMA.F5VerificacionOrdenada or MAIN.fbFMS205.dr.gmModeActual=L1_GEMMA.A1ParadaInicial)
        toggle MAIN.fbFMS205.fbPanel.mdF5Funcion
    Rectangle (1310,422 57x27), "F_1", input disabled if: not MAIN.fbFMS205.dr.cnF4_Planta
        toggle MAIN.fbFMS205.mdEvacuador.F_1.uiValue
    Rectangle (1430,422 57x27), "f1", input disabled if: not MAIN.fbFMS205.dr.cnF4_Planta
        toggle MAIN.fbFMS205.mdEvacuador.f1.uiValue
    Rectangle (10,564 77x27), "Alimentar", input disabled if: MAIN.fbFMS205.dr.gmModeActual<>L1_GEMMA.F5VerificacionOrdenada
        toggle MAIN.fbFMS205.fbPanel.swF5_Alimentar
    Rectangle (90,703 77x27), "Girar", input disabled if: MAIN.fbFMS205.dr.gmModeActual<>L1_GEMMA.F5VerificacionOrdenada
        toggle MAIN.fbFMS205.fbPanel.swF5_Girar
    Rectangle (90,564 77x27), "Situar", input disabled if: MAIN.fbFMS205.dr.gmModeActual<>L1_GEMMA.F5VerificacionOrdenada
        toggle MAIN.fbFMS205.fbPanel.swF5_Situar
    Rectangle (10,634 77x27), "Medir Altura", input disabled if: MAIN.fbFMS205.dr.gmModeActual<>L1_GEMMA.F5VerificacionOrdenada
        toggle MAIN.fbFMS205.fbPanel.swF5_Medir
    Rectangle (90,634 77x27), "Claridad", input disabled if: MAIN.fbFMS205.dr.gmModeActual<>L1_GEMMA.F5VerificacionOrdenada
        toggle MAIN.fbFMS205.fbPanel.swF5_Claridad
    Rectangle (170,634 77x27), "Material", input disabled if: MAIN.fbFMS205.dr.gmModeActual<>L1_GEMMA.F5VerificacionOrdenada
        toggle MAIN.fbFMS205.fbPanel.swF5_Material
    Rectangle (10,664 76x27), "%s", text variable: MAIN.fbFMS205.mdMedidorTapa.strUi, input disabled if: MAIN.fbFMS205.dr.gmModeActual<>L1_GEMMA.F5VerificacionOrdenada
    Rectangle (90,664 77x27), "%s", text variable: MAIN.fbFMS205.mdDetectorFotoelectrico.strUi, input disabled if: MAIN.fbFMS205.dr.gmModeActual<>L1_GEMMA.F5VerificacionOrdenada
    Rectangle (170,664 77x27), "%s", text variable: MAIN.fbFMS205.mdCaptadorInductivo.strUi, input disabled if: MAIN.fbFMS205.dr.gmModeActual<>L1_GEMMA.F5VerificacionOrdenada
    Rectangle (10,603 77x27), "Cargar", input disabled if: MAIN.fbFMS205.dr.gmModeActual<>L1_GEMMA.F5VerificacionOrdenada
        toggle MAIN.fbFMS205.fbPanel.swF5_Cargar
    Rectangle (90,603 77x27), "Evacuar", input disabled if: MAIN.fbFMS205.dr.gmModeActual<>L1_GEMMA.F5VerificacionOrdenada
        toggle MAIN.fbFMS205.fbPanel.swF5_Evacuar
    Rectangle (170,603 77x27), "Descargar", input disabled if: MAIN.fbFMS205.dr.gmModeActual<>L1_GEMMA.F5VerificacionOrdenada
        toggle MAIN.fbFMS205.fbPanel.swF5_Descargar
    Rectangle (170,564 77x27), "Transferir", input disabled if: MAIN.fbFMS205.dr.gmModeActual<>L1_GEMMA.F5VerificacionOrdenada
        toggle MAIN.fbFMS205.fbPanel.swF5_Transferir
    Button (12,741 77x26), "Ejecutar", input disabled if: MAIN.fbFMS205.dr.gmModeActual<>L1_GEMMA.F5VerificacionOrdenada
        tap MAIN.fbFMS205.fbPanel.swF5_Ejecutar
    Button (169,741 77x26), "Visto", input disabled if: MAIN.fbFMS205.dr.gmModeActual<>L1_GEMMA.F5VerificacionOrdenada
        tap MAIN.fbFMS205.fbPanel.swF5_Ack
    Rectangle (1310,452 57x27), "G_1", input disabled if: not MAIN.fbFMS205.dr.cnF4_Planta
        toggle MAIN.fbFMS205.mdEvacuador.G_1.uiValue
    Rectangle (1370,452 57x27), "g0", input disabled if: not MAIN.fbFMS205.dr.cnF4_Planta
        toggle MAIN.fbFMS205.mdEvacuador.g0.uiValue
    Rectangle (1310,482 57x27), "V_1", input disabled if: not MAIN.fbFMS205.dr.cnF4_Planta
        toggle MAIN.fbFMS205.mdEvacuador.V_1.uiValue
    Rectangle (1430,482 57x27), "v1", input disabled if: not MAIN.fbFMS205.dr.cnF4_Planta
        toggle MAIN.fbFMS205.mdEvacuador.v1.uiValue
    Rectangle (1170,512 137x87), "Descarga", input disabled if: not MAIN.fbFMS205.dr.cnF4_Planta
    Rectangle (1310,512 57x27), "H_1", input disabled if: not MAIN.fbFMS205.dr.cnF4_Planta
        toggle MAIN.fbFMS205.mdPickAndPlaceDescarga.HOR.uiValue
    Rectangle (1370,512 57x27), "h0", input disabled if: not MAIN.fbFMS205.dr.cnF4_Planta
        tap MAIN.fbFMS205.mdPickAndPlaceDescarga.h0.uiValue
        toggle MAIN.fbFMS205.mdPickAndPlaceDescarga.h0.uiValue
    Rectangle (1430,512 57x27), "h1", input disabled if: not MAIN.fbFMS205.dr.cnF4_Planta
        toggle MAIN.fbFMS205.mdPickAndPlaceDescarga.h1.uiValue
    Rectangle (1310,542 57x27), "I_1", input disabled if: not MAIN.fbFMS205.dr.cnF4_Planta
        toggle MAIN.fbFMS205.mdPickAndPlaceDescarga.VER.uiValue
    Rectangle (1370,542 57x27), "i0", input disabled if: not MAIN.fbFMS205.dr.cnF4_Planta
        toggle MAIN.fbFMS205.mdPickAndPlaceDescarga.v0.uiValue
    Rectangle (1430,542 57x27), "i1", input disabled if: not MAIN.fbFMS205.dr.cnF4_Planta
        toggle MAIN.fbFMS205.mdPickAndPlaceDescarga.v1.uiValue
    Rectangle (1310,572 57x27), "J_1", input disabled if: not MAIN.fbFMS205.dr.cnF4_Planta
        toggle MAIN.fbFMS205.mdPickAndPlaceDescarga.PIN.uiValue
    Rectangle (1170,602 137x57), "Plato", input disabled if: not MAIN.fbFMS205.dr.cnF4_Planta
    Rectangle (1310,602 57x27), "D_1", input disabled if: not MAIN.fbFMS205.dr.cnF4_Planta
        toggle MAIN.fbFMS205.mdPlatoDivisor.D_1.uiValue
    Rectangle (1370,602 57x27), "d0", input disabled if: not MAIN.fbFMS205.dr.cnF4_Planta
        toggle MAIN.fbFMS205.mdPlatoDivisor.d0.uiValue
    Rectangle (1310,632 57x27), "E_1", input disabled if: not MAIN.fbFMS205.dr.cnF4_Planta
        toggle MAIN.fbFMS205.mdPlatoDivisor.E_1.uiValue
    Rectangle (1170,662 137x117), "Cinta", input disabled if: not MAIN.fbFMS205.dr.cnF4_Planta
    Rectangle (1310,662 57x27), "RUN", input disabled if: not MAIN.fbFMS205.dr.cnF4_Planta
        toggle MAIN.fbFMS205.mdCinta.RUN.uiValue
    Rectangle (1370,662 57x27), "pp", input disabled if: not MAIN.fbFMS205.dr.cnF4_Planta
        toggle MAIN.fbFMS205.mdCinta.pp.uiValue
    Rectangle (1430,662 57x27), "Avanza", colour toggle: MAIN.fbFMS205.mdCinta.RUN.uiValue and Not MAIN.fbFMS205.mdCinta.REV.uiValue, input disabled if: not MAIN.fbFMS205.dr.cnF4_Planta
        tap MAIN.fbFMS205.fbPanel.swF4_Avanza
    Rectangle (1310,692 57x27), "REV", input disabled if: not MAIN.fbFMS205.dr.cnF4_Planta
        toggle MAIN.fbFMS205.mdCinta.REV.uiValue
    Rectangle (1370,692 57x27), "cp0", input disabled if: not MAIN.fbFMS205.dr.cnF4_Planta
        toggle MAIN.fbFMS205.mdCinta.cp0.uiValue
    Rectangle (1431,692 57x27), "Retroc.", colour toggle: MAIN.fbFMS205.mdCinta.RUN.uiValue and MAIN.fbFMS205.mdCinta.REV.uiValue, input disabled if: not MAIN.fbFMS205.dr.cnF4_Planta
        tap MAIN.fbFMS205.fbPanel.swF4_Retroc
    Rectangle (1310,722 57x27), "R_1", input disabled if: not MAIN.fbFMS205.dr.cnF4_Planta
        toggle MAIN.fbFMS205.mdCinta.R_1.uiValue
    Rectangle (1370,722 57x27), "cp1", input disabled if: not MAIN.fbFMS205.dr.cnF4_Planta
        toggle MAIN.fbFMS205.mdCinta.cp1.uiValue
    Rectangle (1310,752 57x27), "S_1", input disabled if: not MAIN.fbFMS205.dr.cnF4_Planta
        toggle MAIN.fbFMS205.mdCinta.S_1.uiValue
    Rectangle (1370,752 57x27), "cp2", input disabled if: not MAIN.fbFMS205.dr.cnF4_Planta
        toggle MAIN.fbFMS205.mdCinta.cp2.uiValue
    Rectangle (11,798 1131x27), "%s", text variable: main.fbFMS205.fbPanel.swMensaje
    Rectangle (1173,797 74x27), "%s", text variable: MAIN.fbFMS205.fbPanel.gmModeName, colour variable: MAIN.fbFMS205.dr.gmModeColor
        p3450524324: MAIN.fbFMS205.dr.gmModeColor
    Rectangle (1250,797 237x27), "%s", text variable: MAIN.fbFMS205.fbPanel.gmModeDescr, colour variable: MAIN.fbFMS205.dr.gmModeColor
        p3450524324: MAIN.fbFMS205.dr.gmModeColor
    Ellipse (12,25 200x200)
    Ellipse (162,105 40x40), "%s", tooltip "%s", text variable: MAIN.fbFMS205.tapas.vstrUi[7], colour variable: MAIN.fbFMS205.tapas.vColorFill[7]
        p2277200375: MAIN.fbFMS205.mdPlatoDivisor.Angulo
        p4168582468: MAIN.fbFMS205.tapas.vstrToolTip[7]
        p55702900: MAIN.fbFMS205.tapas.vColorFont[7]
        p3450524324: MAIN.fbFMS205.tapas.vColorFrame[7]
    Ellipse (141,154 40x40), "%s", tooltip "%s", text variable: MAIN.fbFMS205.tapas.vstrUi[0], colour variable: MAIN.fbFMS205.tapas.vColorFill[0]
        p2277200375: MAIN.fbFMS205.mdPlatoDivisor.Angulo
        p4168582468: MAIN.fbFMS205.tapas.vstrToolTip[0]
        p55702900: MAIN.fbFMS205.tapas.vColorFont[0]
        p3450524324: MAIN.fbFMS205.tapas.vColorFrame[0]
    Ellipse (92,175 40x40), "%s", tooltip "%s", text variable: MAIN.fbFMS205.tapas.vstrUi[1], colour variable: MAIN.fbFMS205.tapas.vColorFill[1]
        p2277200375: MAIN.fbFMS205.mdPlatoDivisor.Angulo
        p4168582468: MAIN.fbFMS205.tapas.vstrToolTip[1]
        p55702900: MAIN.fbFMS205.tapas.vColorFont[1]
        p3450524324: MAIN.fbFMS205.tapas.vColorFrame[1]
    Ellipse (43,154 40x40), "%s", tooltip "%s", text variable: MAIN.fbFMS205.tapas.vstrUi[2], colour variable: MAIN.fbFMS205.tapas.vColorFill[2]
        p2277200375: MAIN.fbFMS205.mdPlatoDivisor.Angulo
        p4168582468: MAIN.fbFMS205.tapas.vstrToolTip[2]
        p55702900: MAIN.fbFMS205.tapas.vColorFont[2]
        p3450524324: MAIN.fbFMS205.tapas.vColorFrame[2]
    Ellipse (22,105 40x40), "%s", tooltip "%s", text variable: MAIN.fbFMS205.tapas.vstrUi[3], colour variable: MAIN.fbFMS205.tapas.vColorFill[3]
        p2277200375: MAIN.fbFMS205.mdPlatoDivisor.Angulo
        p4168582468: MAIN.fbFMS205.tapas.vstrToolTip[3]
        p55702900: MAIN.fbFMS205.tapas.vColorFont[3]
        p3450524324: MAIN.fbFMS205.tapas.vColorFrame[3]
    Ellipse (43,56 40x40), "%s", tooltip "%s", text variable: MAIN.fbFMS205.tapas.vstrUi[4], colour variable: MAIN.fbFMS205.tapas.vColorFill[4]
        p2277200375: MAIN.fbFMS205.mdPlatoDivisor.Angulo
        p4168582468: MAIN.fbFMS205.tapas.vstrToolTip[4]
        p55702900: MAIN.fbFMS205.tapas.vColorFont[4]
        p3450524324: MAIN.fbFMS205.tapas.vColorFrame[4]
    Ellipse (92,35 40x40), "%s", tooltip "%s", text variable: MAIN.fbFMS205.tapas.vstrUi[5], colour variable: MAIN.fbFMS205.tapas.vColorFill[5]
        p2277200375: MAIN.fbFMS205.mdPlatoDivisor.Angulo
        p4168582468: MAIN.fbFMS205.tapas.vstrToolTip[5]
        p55702900: MAIN.fbFMS205.tapas.vColorFont[5]
        p3450524324: MAIN.fbFMS205.tapas.vColorFrame[5]
    Ellipse (141,56 40x40), "%s", tooltip "%s", text variable: MAIN.fbFMS205.tapas.vstrUi[6], colour variable: MAIN.fbFMS205.tapas.vColorFill[6]
        p2277200375: MAIN.fbFMS205.mdPlatoDivisor.Angulo
        p4168582468: MAIN.fbFMS205.tapas.vstrToolTip[6]
        p55702900: MAIN.fbFMS205.tapas.vColorFont[6]
        p3450524324: MAIN.fbFMS205.tapas.vColorFrame[6]
    Image (286,269 853x509), image: ImagePool.img_fms205
    Image (1370,3 111x117), image: ImagePool.img_logo
        p2858320360: sel(MAIN.fbFMS205.dr.gmLocalHost,0,-90)
        OnMouseClick: toggle MAIN.fbFMS205.dr.gmLocalHost
    Image (725,147 418x57), image: ImagePool.img_panel
    Image (101,114 28x30), invisible if: MAIN.fbFMS205.mdPlatoDivisor.Ready, image: VisuSymbols.Symbols.ArrowHalfLeftUp
        p2277200375: MAIN.fbFMS205.mdPlatoDivisor.Angulo
    Image (153,17 32x32), invisible if: MAIN.fbFMS205.mdMedidorTapa.Ready, image: VisuSymbols.Symbols.ArrowBoldDown
    Image (99,5 32x32), invisible if: MAIN.fbFMS205.mdDetectorFotoelectrico.Ready, image: VisuSymbols.Symbols.Download
    Image (25,27 32x32), invisible if: MAIN.fbFMS205.mdCaptadorInductivo.Ready, image: VisuSymbols.Symbols.Download
    Image (15,192 32x32), invisible if: MAIN.fbFMS205.mdEvacuador.Ready, image: VisuSymbols.Symbols.ArrowBoldLeftDown
    Image (94,228 32x32), invisible if: MAIN.fbFMS205.mdPickAndPlaceDescarga.Ready, image: VisuSymbols.Symbols.ArrowBoldDown
    Image (141,232 32x32), invisible if: MAIN.fbFMS205.mdCinta.Ready, image: VisuSymbols.Symbols.ArrowBoldRight
    Meter180 (1171,3 190x98), value: MAIN.fbFMS205.dr.Speed, style: Meter-Meter180-Gray, scale format: %.1f, scale 0..200
    Slider (1180,102 172x31), variable: MAIN.fbFMS205.dr.Speed, scale 1..200
    Rectangle (878,450 89x152), colour variable: MAIN.fbFMS205.mdPickAndPlaceCarga.fbController.colPicFill
        p3450524324: MAIN.fbFMS205.mdPickAndPlaceCarga.fbController.colPicFram
    Rectangle (916,410 56x54), angle 322, colour variable: MAIN.fbFMS205.mdAlimentador.fbController.colPicFill
        p3450524324: MAIN.fbFMS205.mdAlimentador.fbController.colPicFram
    Rectangle (764,277 98x179), angle 4, colour variable: MAIN.fbFMS205.mdMedidorTapa.fbController.colPicFill
        p3450524324: MAIN.fbFMS205.mdMedidorTapa.fbController.colPicFram
    Rectangle (709,330 40x116), colour variable: MAIN.fbFMS205.mdDetectorFotoelectrico.fbController.colPicFill
        p3450524324: MAIN.fbFMS205.mdDetectorFotoelectrico.fbController.colPicFram
    Rectangle (651,338 40x116), angle 353, colour variable: MAIN.fbFMS205.mdCaptadorInductivo.fbController.colPicFill
        p3450524324: MAIN.fbFMS205.mdCaptadorInductivo.fbController.colPicFram
    Rectangle (462,368 174x114), angle 351, colour variable: MAIN.fbFMS205.mdEvacuador.fbController.colPicFill
        p3450524324: MAIN.fbFMS205.mdEvacuador.fbController.colPicFram
    Rectangle (681,547 72x83), colour variable: MAIN.fbFMS205.mdPickAndPlaceDescarga.fbController.colPicFill
        p3450524324: MAIN.fbFMS205.mdPickAndPlaceDescarga.fbController.colPicFram
    Rectangle (521,648 300x99), colour variable: MAIN.fbFMS205.mdCinta.fbController.colPicFill
        p3450524324: MAIN.fbFMS205.mdCinta.fbController.colPicFram
    Ellipse (628,464 195x80), colour variable: MAIN.fbFMS205.mdPlatoDivisor.fbController.colPicFill
        p3450524324: MAIN.fbFMS205.mdPlatoDivisor.fbController.colPicFram
    Rectangle (130,446 97x27), "Probar (F6)", input disabled if: not MAIN.fbFMS205.fbPanel.mdF1Producir
        toggle MAIN.fbFMS205.fbPanel.swF6_Probar
    Rectangle (30,446 97x27), "Finalizar (F3)", input disabled if: not MAIN.fbFMS205.fbPanel.mdF1Producir
        toggle MAIN.fbFMS205.fbPanel.swF3_Finalizar
    Button (10,383 237x26), "Estación"
        toggle MAIN.fbFMS205.fbPanel.mdF1Producir
    Polygon (372,691) (372,691) (390,705) (374,721) (438,708), colour variable: MAIN.fbFMS205.mdCinta.colPicFillSituar
        p3450524324: MAIN.fbFMS205.mdCinta.colPicFramSituar
    Polygon (906,692) (906,692) (924,706) (908,722) (972,709), colour variable: MAIN.fbFMS205.mdCinta.colPicFillTransferir
        p3450524324: MAIN.fbFMS205.mdCinta.colPicFramTransferir
    Lamp1 (1032,534 55x42), variable: MAIN.fbFMS205.mdAlimentador.FM.uiValue, style: Lamp-Lamp1-Red
    PowerSwitch (797,93 45x45), tooltip "Conmutador encendido/apagado", behaviour: TOGGLE, style: Switch-PowerSwitch-Gray
    DipSwitch (736,95 45x45), tooltip "Parada de emergencia (A1)", variable: MAIN.fbFMS205.fbPanel.swPE_Seta, behaviour: TOGGLE, style: Switch-DipSwitch-Red
    PushSwitch (857,95 45x45), tooltip "Pulsador de marcha", variable: MAIN.fbFMS205.fbPanel.SwPM_PulsadorMarcha, behaviour: TAP, style: Switch-PushSwitch-Green
    RotarySwitch (977,95 45x45), tooltip "Selector manual automático (F4)", variable: MAIN.fbFMS205.fbPanel.swSM_SelecAutoManual, behaviour: TOGGLE, style: Switch-RotarySwitch-Gray
    Ellipse (221,55 40x40), "%s", tooltip "%s", text variable: '???', colour variable: colTapFill
        p4168582468: 'Tapa de altura, claridad y color desconocidos'
        p55702900: colTapFont
        p3450524324: colTapFrameSin
        p2738717112: MAIN.fbFMS205.tapas.AlimeY
    Ellipse (220,42 40x40), "%s", tooltip "%s", text variable: 'n', colour variable: colTapFill
        p4168582468: 'Cilindro de carga con n tapas'
        p55702900: colTapFont
        p3450524324: colTapFrameSin
    Lamp1 (857,210 45x45), tooltip "Lámpara de marcha", variable: MAIN.fbFMS205.fbPanel.hwLM_LamparaMarcha, style: Lamp-Lamp1-Green
    Lamp1 (1101,210 47x45), tooltip "Lámpara de alarma", variable: MAIN.fbFMS205.fbPanel.hwLA_LamparaAlarma, style: Lamp-Lamp1-Red
    Lamp1 (1040,210 47x45), tooltip "Lámpara de alarma", variable: TRUE, style: Lamp-Lamp1-Blue
    Image (732,210 45x45), tooltip "Avisador sonoro", invisible if: not MAIN.fbFMS205.fbPanel.hwAS_AvisadorSonoro, image: VisuSymbols.Symbols.loudspeakerLoud
    PushSwitch (917,95 45x45), tooltip "Pulsador de parada", variable: MAIN.fbFMS205.fbPanel.swPS_PulsadorStop, behaviour: TAP, style: Switch-PushSwitch-Green
    PushSwitch (1040,95 45x45), tooltip "Pulsador de inicializar (A6)", variable: MAIN.fbFMS205.fbPanel.swPOC_PulsadorReset, behaviour: TAP, style: Switch-PushSwitch-Green
    Ellipse (221,154 40x40), "%s", tooltip "%s", text variable: '???', invisible if: not MAIN.fbFMS205.tapas.Alimentada, colour variable: colTapFill
        p4168582468: 'Tapa de altura, claridad y color desconocidos'
        p55702900: colTapFont
        p3450524324: colTapFrameSin
        p3560616238: -MAIN.fbFMS205.tapas.CargaX
    Image (186,160 32x32), invisible if: MAIN.fbFMS205.mdPickAndPlaceCarga.Ready, image: VisuSymbols.Symbols.ArrowBoldLeft
    Image (224,115 32x32), invisible if: MAIN.fbFMS205.mdAlimentador.Ready, image: VisuSymbols.Symbols.ArrowBoldDown
        p2175578022: MAIN.fbFMS205.mdPickAndPlaceCarga.fbController.colPicFill
    Ellipse (91,183 40x40), "%s", tooltip "%s", text variable: MAIN.fbFMS205.tapas.Desca_strUi, invisible if: not (MAIN.fbFMS205.mdCinta.TapaDescargada or MAIN.fbFMS205.mdPickAndPlaceDescarga.fbController.Executing), colour variable: MAIN.fbFMS205.tapas.desca_ColorFill
        p4168582468: MAIN.fbFMS205.tapas.Desca_strToolTip
        p55702900: MAIN.fbFMS205.tapas.desca_ColorFont
        p3450524324: MAIN.fbFMS205.tapas.desca_ColorFrame
        p3560616238: MAIN.fbFMS205.tapas.DescaX
        p2738717112: MAIN.fbFMS205.tapas.DescaY
    Rectangle (85,277 50x50)
        p3560616238: MAIN.fbFMS205.tapas.CintaX
    Rectangle (222,266 60x74)
    Ellipse (140,153 8x9)
        p2277200375: MAIN.fbFMS205.mdPlatoDivisor.Angulo
END_VISUALIZATION
